KUKA KRL program: rs.src, rs.dat

--- rs.src ---
&ACCESS RVO
&REL 74
DEF rs(st :OUT)
DECL ST_RS st

st.Q1 = NOT st.RESET1 AND (st.Q1 OR st.SET)

END

GLOBAL DEF sr(st :OUT)
DECL ST_SR st

st.Q1 = (NOT st.RESET AND st.Q1) OR st.SET1

END

--- rs.dat ---
&ACCESS RVO
&REL 74
DEFDAT rs PUBLIC

GLOBAL STRUC ST_RS BOOL SET, RESET1, Q1
GLOBAL STRUC ST_SR BOOL SET1, RESET, Q1

ENDDAT
